(* IEC 61131-3 sources: 2026_Projet_YGO_ExcavatriceDragage/.tmp_conv_test2, 9 files *)

(* ---- E_Mode.st ---- *)
(* =======================================================================
   ⚙️ E_Mode — Modes de marche de la machine
   ───────────────────────────────────────────────────────────────
   🎯 Rôle : Énumération des modes d'exploitation et maintenance
   📄 Doc métier : DOC/AF/AF_Partie-05_Modes_Maintenance_v2.1.md
   ======================================================================= *)
TYPE E_Mode :
    (DISABLE := 0, MAINT_N1 := 1, MAINT_N2 := 2, SEMI_AUTO := 3);
END_TYPE

(* ---- E_State.st ---- *)
(* =======================================================================
   ⚙️ E_State — Phase opérationnelle d'un FB métier (valeurs EXCLUSIVES)
   ───────────────────────────────────────────────────────────────
   🎯 Rôle : Énumération des phases opérationnelles d'un FB métier
   ⚙️ Machine d'état : Un seul état actif à la fois (orthogonal à Error)
   📄 Doc métier : DOC/AF/AF_Partie-03_Contrats_Composants_v2.3.md §3
   ======================================================================= *)

TYPE E_State :
    (DISABLED := 0, INIT := 1, READY := 2, BUSY := 3, DONE := 4, STOPPING := 5, ERROR := 6);
END_TYPE

(* ---- ST_fbJoystick_AxisCmd.st ---- *)
(* =======================================================================
   🕹️ ST_fbJoystick_AxisCmd — Consigne d'axe normalisée (sortie FB_Joystick)
   ───────────────────────────────────────────────────────────────
   🎯 Rôle : Structure de consigne d'axe produite par FB_Joystick.
   📤 Champs : Enable, StartStop, SpeedTgt (%) + StepTgt (palier 1..5) + direction en bits
               (DirectionPositive/Negative, AtNeutral). SpeedTgt reste pour l'IHM, StepTgt pour la logique.
   📄 Doc métier : DOC/AF/AF_Partie-08_Fonction_Joystick_v2.5.md
   ======================================================================= *)

TYPE ST_fbJoystick_AxisCmd :
STRUCT
    // === CONSIGNES DE PILOTAGE AXE ===
    Enable      : BOOL;   // --> [CMD] Autorisation globale pipeline (FALSE=neutralisation, sorties coupees)
    StartStop   : BOOL;   // --> [CMD] Validation de mouvement (TRUE=acceleration, FALSE=deceleration/arret)
    SpeedTgt    : REAL;   // --> [CMD] Vitesse cible non signee (0...100 %, signe/sens donné par Direction) - IHM
    StepTgt     : INT;    // --> [CMD] Palier de vitesse (1..5, 0=arret) - logique/limitations (derive de SpeedTgt)
    DirectionNegative   : BOOL;   // --> [CMD] Direction joystick ou intension de gestuelle
    DirectionPositive   : BOOL;   // --> [CMD] Direction joystick ou intension de gestuelle
    AtNeutral   : BOOL;   // --> [CMD] TRUE si axes en zone morte (position centrale)

    // === MONITORING IHM (derive des bits ci-dessus, jamais lu en interlock) ===
    Direction   : INT;   // <-- [STAT] Sens -1=Rev / 0=Neutre / +1=Fwd (anim IHM fleche ; lu aussi logique treuils PRG_04)
    Deflection  : INT;   // <-- [STAT] Deflexion signee -100..+100 % (anim IHM jauge/barre)
END_STRUCT
END_TYPE

(* ---- FB_Acquisition_Preflight.st ---- *)
(* =======================================================================
   📊 FB_Acquisition_Preflight — Verdict passif machine arrêtée
   ───────────────────────────────────────────────────────────────
   🎯 Rôle : Verdict passif de qualification E/S machine arrêtée (16 contrôles)
   🔒 Polarité : Observateur pur (aucun SafeStop, PowerCutOff ou ordre machine)
   📄 Doc métier : DOC/AF/AF_Partie-06_Acquisition_Qualification_IO_v2.4.md §6
   ======================================================================= *)
FUNCTION_BLOCK FB_Acquisition_Preflight
VAR_INPUT
    // === COMMANDES & ETATS MACHINE ===
    Execute                 : BOOL; // --> [CMD] Lancement du verdict (front montant)
    MachineIsStill          : BOOL; // --> [HW]  Machine a l'arret complet (vitesse nulle)

    // === ETATS FREINS & CONTACTEURS ===
    M1BrakeApplied          : BOOL; // --> [HW]  Frein M1 serre
    M2BrakeApplied          : BOOL; // --> [HW]  Frein M2 serre
    M3BrakeApplied          : BOOL; // --> [HW]  Frein M3 serre
    M1ContactorsReleased    : BOOL; // --> [HW]  Contacteurs M1 retombes
    M2ContactorsReleased    : BOOL; // --> [HW]  Contacteurs M2 retombes

    // === PROTECTION THERMIQUE & RESEAU ===
    M1ThermalOk             : BOOL; // --> [HW]  Thermique moteur M1 OK
    M2ThermalOk             : BOOL; // --> [HW]  Thermique moteur M2 OK
    BrakeThermalOk          : BOOL; // --> [HW]  Thermique freins OK
    PhaseRotationOk         : BOOL; // --> [HW]  Ordre des phases reseau OK

    // === CAPTEURS & CHAINE DE SECURITE ===
    SlackCableTensioned     : BOOL; // --> [HW]  Cable M2 tendu (anti-mou)
    M3SensorWordIncoherent  : BOOL; // --> [HW]  Incoherence mot capteurs M3
    EmergencyChainClosed    : BOOL; // --> [SAFE] Chaine d'arret d'urgence fermee
    PowerContactorEngaged   : BOOL; // --> [HW]  Contacteur de puissance enclenche

    // === CODEURS & HOMING ===
    EncoderM1Operational    : BOOL; // --> [HW]  Codeur M1 operationnel
    EncoderM2Operational    : BOOL; // --> [HW]  Codeur M2 operationnel
    HomedM1                 : BOOL; // --> [HW]  Homing M1 effectue
    HomedM2                 : BOOL; // --> [HW]  Homing M2 effectue
    M1PositionInBounds      : BOOL; // --> [HW]  Position M1 dans les bornes
    M2PositionInBounds      : BOOL; // --> [HW]  Position M2 dans les bornes
END_VAR
VAR_OUTPUT
    // === ETATS ET DIAGNOSTIC ===
    PreflightOk             : BOOL; // <-- [STAT] Verdict preflight OK (aucun defaut)
    PreflightDone           : BOOL; // <-- [STAT] Verdict preflight termine
    PreflightBusy           : BOOL; // <-- [STAT] Diagnostic preflight en cours
    PreflightErrorId        : WORD; // <-- [DIAG] Masque de defauts preflight (16 bits)
END_VAR
VAR
    // === TRIGGERS & ETATS INTERNES ===
    ExecuteEdge             : R_TRIG;       // . [LOC] Trigger front montant Execute
    RequestPending          : BOOL;         // . [LOC] Demande de verdict en attente
END_VAR

ExecuteEdge(CLK := Execute);
RequestPending := RequestPending OR ExecuteEdge.Q;
PreflightBusy := RequestPending AND NOT MachineIsStill;
IF NOT MachineIsStill THEN PreflightDone := FALSE; RETURN; END_IF;
IF NOT RequestPending THEN RETURN; END_IF;

PreflightErrorId := 0;
(* bit0..2 frein M1/M2/M3 serré; bit3..4 contacteurs M1/M2 retombés;
   bit5..6 thermique M1/M2 OK; bit7 thermique frein OK; bit8 phases OK;
   bit9 câble M2 tendu; bit10 mot M3 cohérent; bit11 contacteur sans chaîne;
   bit12..13 codeur M1/M2 opérationnel; bit14..15 homé et position bornée M1/M2. *)
IF NOT M1BrakeApplied THEN PreflightErrorId := PreflightErrorId OR 16#0001; END_IF;
IF NOT M2BrakeApplied THEN PreflightErrorId := PreflightErrorId OR 16#0002; END_IF;
IF NOT M3BrakeApplied THEN PreflightErrorId := PreflightErrorId OR 16#0004; END_IF;
IF NOT M1ContactorsReleased THEN PreflightErrorId := PreflightErrorId OR 16#0008; END_IF;
IF NOT M2ContactorsReleased THEN PreflightErrorId := PreflightErrorId OR 16#0010; END_IF;
IF NOT M1ThermalOk THEN PreflightErrorId := PreflightErrorId OR 16#0020; END_IF;
IF NOT M2ThermalOk THEN PreflightErrorId := PreflightErrorId OR 16#0040; END_IF;
IF NOT BrakeThermalOk THEN PreflightErrorId := PreflightErrorId OR 16#0080; END_IF;
IF NOT PhaseRotationOk THEN PreflightErrorId := PreflightErrorId OR 16#0100; END_IF;
IF NOT SlackCableTensioned THEN PreflightErrorId := PreflightErrorId OR 16#0200; END_IF;
IF M3SensorWordIncoherent THEN PreflightErrorId := PreflightErrorId OR 16#0400; END_IF;
IF PowerContactorEngaged AND NOT EmergencyChainClosed THEN PreflightErrorId := PreflightErrorId OR 16#0800; END_IF;
IF NOT EncoderM1Operational THEN PreflightErrorId := PreflightErrorId OR 16#1000; END_IF;
IF NOT EncoderM2Operational THEN PreflightErrorId := PreflightErrorId OR 16#2000; END_IF;
IF NOT HomedM1 OR NOT M1PositionInBounds THEN PreflightErrorId := PreflightErrorId OR 16#4000; END_IF;
IF NOT HomedM2 OR NOT M2PositionInBounds THEN PreflightErrorId := PreflightErrorId OR 16#8000; END_IF;

PreflightOk := (PreflightErrorId = 0); PreflightDone := TRUE; RequestPending := FALSE;
END_FUNCTION_BLOCK

(* ---- FB_Brake.st ---- *)
(* =======================================================================
   🛡️ FB_Brake — Séquence frein à manque de courant (temps physiques)
   ───────────────────────────────────────────────────────────────
   🎯 Rôle : Gestion temporisée ouverture/fermeture frein à manque de courant
   🔒 Polarité : Sécurité positive (BrakeCmd=FALSE = frein collé au repos)
   🔌 Interface : Double vérification retour contacteur (ST_ContactorCheck)
   📄 Doc métier : DOC/AF/AF_Partie-10_Fonction_Winch_v2.1.md §3
   ======================================================================= *)
FUNCTION_BLOCK FB_Brake
VAR_INPUT
    // === COMMANDES ET CONSIGNES ===
    Enable                  : BOOL;               // --> [CMD]  Autorisation generale (FALSE = frein colle)
    Reset                   : BOOL;               // --> [CMD]  Acquittement defaut (front)
    MovementRequested       : BOOL;               // --> [CMD]  Demande de mouvement (sens+palier actifs)

    // === RETOURS MATERIELS & SIMULATION ===
    ContactorFeedback       : BOOL;               // --> [HW]   Retour contacteur frein (TRUE = relache/ouvert)
    BypassContactorCheck    : BOOL;               // --> [TST]  Bypass controle contacteur (simu)

    // === TEMPORISATIONS ET REGLAGES ===
    DelayContactClose       : TIME := T#100ms;    // --> [CFG]  Temps de fermeture contacteur de puissance
    DelayMagnetise          : TIME := T#300ms;    // --> [CFG]  Delai magnetisation moteur avant ouverture frein
    DelayMotorDecel         : TIME := T#500ms;    // --> [CFG]  Delai deceleration avant collage frein
    FeedbackTimeout         : TIME := T#1s;       // --> [CFG]  Delai max coherence commande/retour frein
END_VAR
VAR_OUTPUT
    // === ETATS IEC & DERIVATION ===
    Ready                   : BOOL;               // <-- [STAT] FB pret a fonctionner
    // 🧩 Statut transverse (forme cible ST_Fault)
    Fault                   : ST_Fault;

    // === COMMANDES ET CONFIRMATIONS ===
    BrakeCmd                : BOOL;               // <-- [ACT]  Commande bobine frein (TRUE = relache/ouvert)
    BrakeCommandOpenConfirmed : BOOL;            // <-- [STAT] Confirmation ouverture frein pour verrous
    ContactorCheck          : ST_ContactorCheck;  // <-- [DIAG] Diagnostic detaille retour contacteur
END_VAR
VAR
    // === TRIGGERS ET DETECTION FRONTS ===
    ResetEdge               : R_TRIG;             // . [LOC]  Detecteur front acquittement
    BypassEdge              : R_TRIG;             // . [LOC]  Detecteur front activation bypass

    // === TEMPORISATEURS INTERNES ===
    TonMagnetise            : TON;                // . [LOC]  Temporisation avant relachement frein
    TonDecel                : TON;                // . [LOC]  Temporisation avant collage frein
    TonFeedback             : TON;                // . [LOC]  Timeout de coherence commande/retour

    // === GESTION DES DEFAUTS ===
    ContactorIncoherentError: BOOL;               // . [LOC]  Défaut mémorisé incohérence contacteur
    instFault               : FB_FaultCore;       // * [INST] Socle de défaut
    instCauses              : ARRAY[0..15] OF ST_FaultCause; // . [LOC] Table des causes nommées
END_VAR

// === IMPLEMENTATION ===

// 🔑 1. FRONTS
ResetEdge(CLK := Reset);
BypassEdge(CLK := BypassContactorCheck);

// Acquittement des drapeaux contacteur
IF ResetEdge.Q OR BypassContactorCheck THEN
    ContactorIncoherentError := FALSE;
    ContactorCheck.StuckClosed := FALSE;
    ContactorCheck.StuckOpen   := FALSE;
END_IF;

// 🛑 2. GATE — pas d'Enable = frein collé (sécurité positive), aucune temporisation en cours
IF NOT Enable THEN
    TonMagnetise(IN := FALSE, PT := DelayMagnetise + DelayContactClose);
    TonDecel(IN := FALSE, PT := DelayMotorDecel);
    TonFeedback(IN := FALSE, PT := FeedbackTimeout);
    BrakeCmd := FALSE;
    Ready := FALSE;
    ContactorCheck.Command := FALSE;          // 📊 Neutralisation : miroir de BrakeCmd := FALSE
    ContactorCheck.Feedback := ContactorFeedback; // 📊 Neutralisation : miroir entrée physique
    BrakeCommandOpenConfirmed := FALSE;       // 🛡️ Fail-Safe : frein commandé fermé hors Enable

    // Évaluation du socle de défaut sous neutralisation (permet acquittement Reset hors Enable)
    instCauses[0].Active   := FALSE;
    instCauses[0].Latching := TRUE;
    instCauses[0].Texte    := 'Incoherence retour contacteur frein';
    instFault(Enable := FALSE, Reset := Reset, Causes := instCauses);
    Fault := instFault.Fault;
    RETURN;
END_IF;

// 🛠️ 3. SÉQUENCE TEMPORISÉE (démarrage vs arrêt)
IF MovementRequested THEN
    TonDecel(IN := FALSE, PT := DelayMotorDecel);
    TonMagnetise(IN := TRUE, PT := DelayMagnetise + DelayContactClose);
    IF TonMagnetise.Q THEN
        BrakeCmd := TRUE;              // ✅ Contacteur + magnétisation acquis → relâche
    ELSE
        BrakeCmd := FALSE;             // ⏳ Encore collé pendant la magnétisation
    END_IF;
ELSE
    // Sécurité positive : fermeture immédiate du frein (collé) dès que les contacteurs de sens s'ouvrent
    TonMagnetise(IN := FALSE, PT := DelayMagnetise + DelayContactClose);
    TonDecel(IN := FALSE, PT := DelayMotorDecel);
    BrakeCmd := FALSE;                 // Fermeture immédiate
END_IF;

// 🔍 4. DOUBLE VÉRIFICATION RETOUR CONTACTEUR (ST_ContactorCheck)
ContactorCheck.Command := BrakeCmd;
ContactorCheck.Feedback := ContactorFeedback;

// ContactorFeedback est dans le MÊME sens que BrakeCmd (TRUE = relâché = frein ouvert).
TonFeedback(IN := (BrakeCmd <> ContactorFeedback), PT := FeedbackTimeout);
IF NOT BypassContactorCheck THEN
    IF TonFeedback.Q THEN
        ContactorCheck.StuckClosed := (BrakeCmd AND NOT ContactorFeedback);
        ContactorCheck.StuckOpen   := (NOT BrakeCmd AND ContactorFeedback);
        ContactorIncoherentError   := TRUE;
    END_IF;
END_IF;

// 🚨 5. SOCLE DÉFAUT & SORTIE SÛRE
instCauses[0].Active   := NOT BypassContactorCheck AND (ContactorCheck.StuckClosed OR ContactorCheck.StuckOpen OR (TonFeedback.Q AND (BrakeCmd <> ContactorFeedback)));
instCauses[0].Latching := TRUE;
instCauses[0].Texte    := 'Incoherence retour contacteur frein';

instFault(Enable := Enable, Reset := Reset, Causes := instCauses);
Fault := instFault.Fault;

Ready := Enable AND NOT Fault.Latched;

// Sortie sûre immédiate
IF Fault.Error OR Fault.Latched THEN
    BrakeCmd := FALSE;
END_IF;

// 📤 6. CONFIRMATION OUVERTURE FREIN
IF BypassContactorCheck THEN
    BrakeCommandOpenConfirmed := BrakeCmd;
ELSE
    BrakeCommandOpenConfirmed := ContactorFeedback AND NOT Fault.Latched;  (* TRUE = frein ouvert = desserrage confirmé *)
END_IF;
END_FUNCTION_BLOCK

(* ---- FB_CycleTime.st ---- *)
(* =======================================================================
   ⚙️ FB_CycleTime — Mesure du temps de cycle réel de la tâche
   ───────────────────────────────────────────────────────────────
   🎯 Rôle : Calcul du dt réel entre deux exécutions successives
   ⚙️ Calcul : Delta horloge système TIME() converti en secondes
   🛡️ Robustesse : dt borné (0 < dt <= CST_MaxCycleDeltaMs) sinon valeur de secours —
      neutralise les artefacts de rebouclage TIME() (49,7 j) et de reprise (online-change, debug)
   📄 Doc métier : DOC/AF/AF_Partie-03_Contrats_Composants/FB_CycleTime_v1.0.md
   ======================================================================= *)
FUNCTION_BLOCK FB_CycleTime
VAR_INPUT
    // === REGLAGES DE SECOURS ===
    DefaultValueS           : REAL := 0.004;      // --> [CFG] Valeur de secours par defaut (ex: 4ms = 0.004s)
END_VAR
VAR_OUTPUT
    // === MESURE ET DIAGNOSTIC ===
    CycleTimeS              : REAL;               // <-- [DIAG] Temps ecoule reel calcule (secondes)
END_VAR
VAR
    // === HORLOGE ET MEMOIRE TEMPORELLE ===
    TimeCurrent             : TIME;               // . [LOC] Temps systeme actuel
    TimeLast                : TIME;               // . [LOC] Empreinte de temps du cycle precedent
    DeltaTimeMs             : UDINT;              // . [LOC] Ecart brut calcule (ms)
    InitDone                : BOOL;               // . [LOC] Drapeau d'initialisation du premier cycle
END_VAR
VAR CONSTANT
    // === BORNE HAUTE DU DELTA DE CYCLE ===
    CST_MaxCycleDeltaMs     : UDINT := 1000;      // Plafond physique du dt entre deux scans (ms) : au-dela -> valeur de secours
END_VAR

// 1. ACQUISITION DU TEMPS SYSTÈME
TimeCurrent := TIME();

// 2. INITIALISATION UNIQUE AU PREMIER CYCLE
IF NOT InitDone THEN
    TimeLast := TimeCurrent;
    InitDone := TRUE;
    CycleTimeS := DefaultValueS;
    RETURN;
END_IF;

// 3. CALCUL DU DELTA EN MILLISECONDES
DeltaTimeMs := TIME_TO_UDINT(TimeCurrent - TimeLast);

// 4. CONVERSION EN SECONDES, AVEC DOUBLE BORNAGE DU DELTA
//
// TIME() est un compteur systeme 32 bits en millisecondes depuis le demarrage de
// l'automate. Il n'est PAS absolu : il reboucle a 0 tous les 2^32 ms (~49,7 jours).
// La soustraction TimeCurrent - TimeLast est modulo 2^32 : au passage du rebouclage,
// tant que l'ecart reel entre deux scans reste < 49,7 j (toujours vrai a 10 ms),
// DeltaTimeMs reste correct. Le rebouclage seul n'est donc pas le risque principal.
//
// Le vrai risque est un DeltaTimeMs REELLEMENT > CST_MaxCycleDeltaMs : reprise apres
// un online-change, sortie d'un point d'arret / pas-a-pas debug, ou fenetre du
// rebouclage TIME(). Le chien de garde tache (200 ms, sensibilite 1) borne deja les
// gels en fonctionnement ; ce plafond couvre les cas hors surveillance.
// Un dt aberrant publie tel quel donnerait un CycleTimeS enorme, propage en un seul
// scan dans les rampes de vitesse et les integrateurs de position/frein -> saut
// physique. Fail-safe : hors de la plage nominale (0 < dt <= plafond), on publie la
// valeur de secours DefaultValueS au lieu de l'artefact. Pas de redemarrage auto.
//
// Borne basse dt = 0 (anti-zero, ex. premier appel du scan) et borne haute
// dt > CST_MaxCycleDeltaMs (anti-artefact) partagent la meme branche de secours.
IF (DeltaTimeMs > 0) AND (DeltaTimeMs <= CST_MaxCycleDeltaMs) THEN
    CycleTimeS := UDINT_TO_REAL(DeltaTimeMs) / 1000.0;
ELSE
    CycleTimeS := DefaultValueS;
END_IF;

// 5. ARCHIVAGE POUR LE PROCHAIN CYCLE
TimeLast := TimeCurrent;
END_FUNCTION_BLOCK

(* ---- FB_FaultCore.st ---- *)
(* =======================================================================
   🧩 FB_FaultCore — Socle de remplissage de ST_Fault (vue live + vue latchée)
   ───────────────────────────────────────────────────────────────
   🎯 Rôle : à partir d'une LISTE de causes en clair (ARRAY[0..15] OF
      ST_FaultCause), produire la brique ST_Fault :
        • Error / ErrorId   : vue LIVE, suit les causes Active, retombe seule.
        • Latched / LatchedId: vue LATCHÉE, chaque bit figé à l'apparition d'une
          cause `Active AND Latching`, conservé jusqu'au front Reset.
   🔒 Sécurité :
      - interlock TOUJOURS sur `Causes[i].Active` (cause brute), jamais sur le latch.
      - Reset TOUJOURS effectif, jamais conditionné (std §9) — agit même Enable=FALSE.
      - Latching=FALSE → cause visible en LIVE seulement (fail-safe : reste visible).
      - un défaut laté non acquitté reste publié même FB désactivé (pas d'effacement
        silencieux sur bascule Enable OFF→ON sans Reset).
      - une cause à acquitter réapparue re-arme son bit (ré-alarme).
   🧬 Un seul socle, réutilisé par tout FB `standard` qui expose un ST_Fault.
      Pas de State, pas de Warning, pas de texte — hors périmètre de ce socle.
   📄 Doc : DOC/STDS/CODE_QUALITY_STANDARDS.md §2quinquies / §9
   ======================================================================= *)

FUNCTION_BLOCK FB_FaultCore
VAR_INPUT
    Enable  : BOOL;                          // --> [CMD] Autorisation générale du FB porteur
    Reset   : BOOL;                          // --> [CMD] Front d'acquittement (jamais conditionné, §9)
    Causes  : ARRAY[0..15] OF ST_FaultCause; // --> [CMD] Liste des causes en clair (Active / Latching / Texte)
END_VAR
VAR_OUTPUT
    Ready   : BOOL;                          // <-- [STAT] FB porteur autorisé (= Enable)
    Fault   : ST_Fault;                      // <-- [DIAG] Brique défaut (mappée 1:1 sur la sortie du FB porteur)
END_VAR
VAR
    ResetEdge : R_TRIG;                      // . [LOC] Front montant Reset
    Latch     : ARRAY[0..15] OF BOOL;        // . [LOC] Bit laté par cause, jusqu'au Reset
    i         : INT;                         // . [LOC] Index de parcours de la liste
END_VAR

// Front Reset : efface tous les latches. Jamais conditionné, agit même Enable=FALSE (§9).
Ready := Enable;
ResetEdge(CLK := Reset);
IF ResetEdge.Q THEN
    FOR i := 0 TO 15 DO Latch[i] := FALSE; END_FOR;
END_IF;

// Bitfield des causes présentes MAINTENANT. Retombe seule à 0 quand les causes disparaissent.
// Non évaluée si Enable=FALSE (pas de lecture de cause hors autorisation).
Fault.ErrorId := 0;
IF Enable THEN
    FOR i := 0 TO 15 DO
        IF Causes[i].Active THEN
            Fault.ErrorId := Fault.ErrorId OR SHL(WORD#1, INT_TO_DWORD(i));
        END_IF;
    END_FOR;
END_IF;
Fault.Error := (Fault.ErrorId <> 0);

// Une cause Active ET Latching arme son bit ; le bit reste jusqu'au front Reset (§1),
// même si la cause disparaît. Réapparition => ré-armement (ré-alarme).
IF Enable THEN
    FOR i := 0 TO 15 DO
        IF Causes[i].Active AND Causes[i].Latching THEN
            Latch[i] := TRUE;
        END_IF;
    END_FOR;
END_IF;

// Toujours publiée, y compris Enable=FALSE : un défaut non acquitté reste visible.
Fault.LatchedId := 0;
FOR i := 0 TO 15 DO
    IF Latch[i] THEN
        Fault.LatchedId := Fault.LatchedId OR SHL(WORD#1, INT_TO_DWORD(i));
    END_IF;
END_FOR;
Fault.Latched := (Fault.LatchedId <> 0);

END_FUNCTION_BLOCK

(* ---- FB_Filter.st ---- *)
(* =======================================================================
   ⚙️ FB_Filter — Filtre passe-bas premier ordre (PT1 numérique)
   ───────────────────────────────────────────────────────────────
   🎯 Rôle : Filtre exponentiel discret y[k] = a*x[k] + (1-a)*y[k-1]
             avec a = CycleTimeS / (T + CycleTimeS). Pass-through si T=0 ou Cycle=0.
   📄 Domaine : CODE/A_COMMUN (fonction de filtrage générale)
   ======================================================================= *)

FUNCTION_BLOCK FB_Filter
VAR_INPUT
    // === CONSIGNES DE PILOTAGE & CONFIGURATION ===
    ValueIn    : REAL;  // --> [CMD] Valeur brute a filtrer
    TimeConst  : TIME;  // --> [CFG] Constante de temps du filtre (ex: T#200ms)
    CycleTimeS : REAL;  // --> [CFG] Temps de cycle reel de la tache en secondes (ex: 0.02)
END_VAR
VAR_OUTPUT
    // === SORTIES LISSÉES ===
    ValueOut   : REAL;  // <-- [STAT] Valeur lissee par filtre PT1
END_VAR
VAR
    // === VARIABLES LOCALES INTERNES ===
    T          : REAL;  // . [LOC]  Constante de temps convertie en secondes
    Alpha      : REAL;  // . [LOC]  Facteur d'attenuation du filtre exponentiel
END_VAR

T := TIME_TO_REAL(TimeConst) / 1000.0; // ms → s

IF T <= 0.0 OR CycleTimeS <= 0.0 THEN
    ValueOut := ValueIn;
ELSE
    Alpha    := CycleTimeS / (T + CycleTimeS);
    ValueOut := Alpha * ValueIn + (1.0 - Alpha) * ValueOut;
END_IF;
END_FUNCTION_BLOCK

(* ---- FB_Ramp.st ---- *)
(* =======================================================================
   ⚙️ FB_Ramp — Rampe d'accélération et décélération asymétrique
   ───────────────────────────────────────────────────────────────
   🎯 Rôle : Limitation de variation anti-à-coups (%/s) sur signal analogique
   🔒 Polarité : Distingue l'éloignement de zéro (Accel) et le retour à zéro (Decel)
   📄 Doc métier : DOC/AF/AF_Partie-11_Fonction_Translation_v2.3.md §1 (TC-P11-040)
   ======================================================================= *)
FUNCTION_BLOCK FB_Ramp
VAR_INPUT
    // === CONSIGNES ET TAUX DE RAMPE ===
    Target                  : REAL;               // --> [CMD] Valeur cible visee (-100.0..+100.0 %)
    AccelRate               : REAL;               // --> [CFG] Taux d'acceleration (%/s)
    DecelRate               : REAL;               // --> [CFG] Taux de deceleration (%/s)
    CycleTimeS              : REAL;               // --> [CFG] Temps de cycle reel en secondes (dt)
END_VAR
VAR_OUTPUT
    // === VALEUR RAMPEE ===
    Current                 : REAL;               // <-- [STAT] Valeur courante amortie (-100.0..+100.0 %)
END_VAR
VAR
    // === CALCULS INTERNES ===
    StepX                   : REAL;               // . [LOC] Pas de variation pour le cycle courant
    TargetLimited           : REAL;               // . [LOC] Cible bornee a [-100.0, +100.0]
END_VAR

// Détection du comportement (Accélération vs Décélération)
// Classification par CÔTÉ DE ZÉRO + sens de déplacement, plus par signe brut de Target seul
// (robuste à une traversée de zéro rapide).
// 🛡️ Garde-fou : la rampe ne sort jamais de la plage normalisée ±100 %.
TargetLimited := LIMIT(-100.0, Target, 100.0);
Current := LIMIT(-100.0, Current, 100.0);

IF (Current >= 0.0 AND TargetLimited >= Current) OR (Current <= 0.0 AND TargetLimited <= Current) THEN
    StepX := AccelRate * CycleTimeS; // S'éloigne du zéro (reste du même côté, va plus loin)
ELSE
    StepX := DecelRate * CycleTimeS; // Retourne vers zéro, ou le traverse vers l'autre signe
END_IF;

// Application de la rampe
IF Current < TargetLimited THEN
    Current := Current + StepX;
    IF Current > TargetLimited THEN Current := TargetLimited; END_IF;
ELSIF Current > TargetLimited THEN
    Current := Current - StepX;
    IF Current < TargetLimited THEN Current := TargetLimited; END_IF;
END_IF;

// 🛡️ Limitation finale : même une valeur d'état déjà corrompue reste bornée.
Current := LIMIT(-100.0, Current, 100.0);
END_FUNCTION_BLOCK
